// TIA Portal V20 export
DATA_BLOCK "DB_ConveyorParameters"   // DB26
// stored: Access Published, MemoryReserve 100, Namespace EmptyLine
   VAR
      Line : Struct
         EmptyLine : Struct
            Conveyor : Array[_.minEmptyLine.._.maxEmptyLine] of "Global.ConveyorParameters";
            Mabs { S7_SetPoint := 'True'} : Array[_."J1.6.1".._."J1.6.2"] of "Global.MABS_Parameters";
         END_STRUCT;
      END_STRUCT;
   END_VAR
BEGIN
END_DATA_BLOCK
